///EL2202 | XFC, 2-channel digital output terminal 24 V DC, TON/TOFF 1 µs, push-pull outputs, tri-state
FUNCTION_BLOCK EL2202_v0_00

END_FUNCTION_BLOCK

(* stored: Version 1.1.0.1, ProductVersion 3.1.4022.6
   POU EL2202_v0_00: Id {9faa20a4-7a9a-4969-913b-a50e4ab982b9}, SpecialFunc None *)
